(* IEC 61131-3 sources: AXOpen/src/data/tests/AXOpen.Data.Tests_L1/ax/src/FragmentData, 2 files *)

(* ---- Context.st ---- *)
USING AXOpen.Core;
using AXOpen.Data;

NAMESPACE Tests_L1.FragmentData

    {S7.extern=ReadWrite}
    CLASS PUBLIC FragmentDataContext EXTENDS AXOpen.Core.AxoContext
        VAR PUBLIC
            _rootObject :   AxoObject;

            DataManager : Tests_L1.FragmentData.FragmentProcessDataManager;
        END_VAR

        METHOD OVERRIDE Main
            THIS.InitializeRootObject(_rootObject);
            DataManager.Run(_rootObject);
        END_METHOD
    END_CLASS

END_NAMESPACE

(* ---- FragmentDataManager.st ---- *)
USING AXOpen.Core;
USING AXOpen.Data;

NAMESPACE Tests_L1.FragmentData

    {S7.extern=ReadWrite}
    CLASS PUBLIC FragmentProcessDataManager EXTENDS AXOpen.Data.AxoDataFragmentExchange
        VAR PUBLIC

            {#ix-attr:[AXOpen.Data.AxoDataFragmentAttribute]}
            EntityHeader : Tests_L1.SharedEntityHeaderManager;

            {#ix-attr:[AXOpen.Data.AxoDataFragmentAttribute]}
            Station :  Tests_L1.StationdataManager;

        END_VAR
    END_CLASS

END_NAMESPACE
